(* Logix 5000 project; controller Proyecto_FRI vendor 1 type 14 code 156 rev 30.11; software revision 30.00 *)

TASK MainTask (continuous, watchdog 500 ms) : MainProgram

MODULES
   Local : vendor 1 type 14 code 156 (Compact 0, rev 30.11)
      INPUTS : 1769-IQ16 (Compact 4, rev 1.1, Input RPI 20 ms)
      OUTPUTS : vendor 1 type 7 code 86 (Compact 5, rev 2.1, Output RPI 20 ms)
END_MODULES

PROGRAM MainProgram   (* main routine MainRoutine *)
VAR
   BANDA : BOOL;
   BR1_RDY : ALIAS FOR Local:4:I.Data.1;   // Brazo 1 termina rutina
   BR2_RDY : ALIAS FOR Local:4:I.Data.2;   // Brazo 2 termina rutina
   FIN : BOOL;
   INICIO : BOOL;
   PARA : BOOL;
   START : BOOL;
   STOP : BOOL;
   STP_BANDA : ALIAS FOR Local:4:I.Data.0;   // Final carrera Banda
   STR_BANDA : ALIAS FOR Local:5:O.Data.0;   // Inicia la banda
   STR_BR1_1 : ALIAS FOR Local:5:O.Data.1;
   STR_BR1_2 : ALIAS FOR Local:5:O.Data.2;
   STR_BR2 : ALIAS FOR Local:5:O.Data.3;
END_VAR

ROUTINE MainRoutine   (* ladder *)
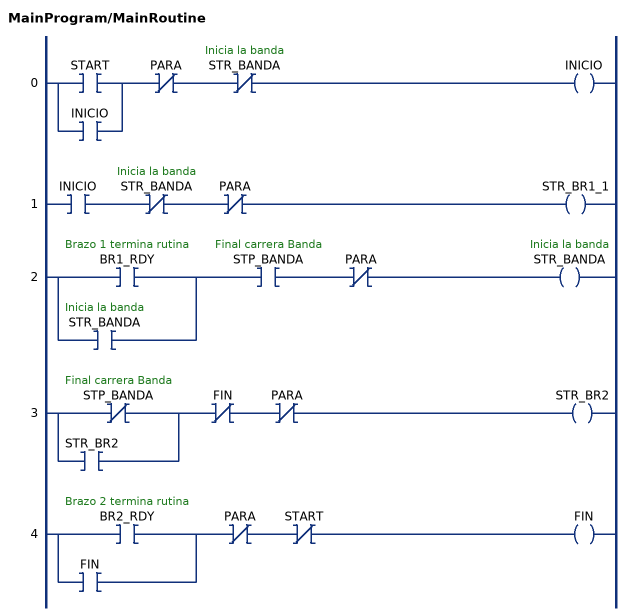
   0: [XIC(START) ,XIC(INICIO) ]XIO(PARA)XIO(STR_BANDA)OTE(INICIO);
   1: XIC(INICIO)XIO(STR_BANDA)XIO(PARA)OTE(STR_BR1_1);
   2: [XIC(BR1_RDY) ,XIC(STR_BANDA) ]XIC(STP_BANDA)XIO(PARA)OTE(STR_BANDA);
   3: [XIO(STP_BANDA) ,XIC(STR_BR2) ]XIO(FIN)XIO(PARA)OTE(STR_BR2);
   4: [XIC(BR2_RDY) ,XIC(FIN) ]XIO(PARA)XIO(START)OTE(FIN);
END_ROUTINE
END_PROGRAM
